{attribute addProperty BoxType "EK1100-0000-0018"}
{attribute addProperty Id "Beckhoff_EM7xxxEK1122Beckhoff_EM7xxxEK1122_7F196951162A_0001_EM7004_0000_9995EM7004_03A980A573692A_0002_EM7004_0000_9996EM7004_78FC6930920115A_0003_EM7004_0000_9997EM7004_78FC6930920115A_0004_EM7004_0000_0016EM7004_A38AEEB0952119A_0005_EM7004_0000_0017EM7004_1DEDE50054468A_0006_EM7004_0000_0018EM7004_1DEDE50054468"}
{attribute addProperty CRC "2403096270"}
{attribute addProperty SizeInBites "4632"}
{attribute addProperty SizeInBytes "579"}
TYPE Beckhoff_EM7xxx_8F3C56CE EXTENDS EK1100_179A0949 :
STRUCT
	{attribute addProperty Name "Beckhoff_EM7xxxEK1122"}
	Beckhoff_EM7xxxEK1122 : Beckhoff_EM7xxxEK1122_7F196951;
	{attribute addProperty Name "A_0001_EM7004_0000_9995"}
	A_0001_EM7004_0000_9995 : EM7004_03A980A5;
	{attribute addProperty Name "A_0002_EM7004_0000_9996"}
	A_0002_EM7004_0000_9996 : EM7004_78FC6930;
	{attribute addProperty Name "A_0003_EM7004_0000_9997"}
	A_0003_EM7004_0000_9997 : EM7004_78FC6930;
	{attribute addProperty Name "A_0004_EM7004_0000_0016"}
	A_0004_EM7004_0000_0016 : EM7004_A38AEEB0;
	{attribute addProperty Name "A_0005_EM7004_0000_0017"}
	A_0005_EM7004_0000_0017 : EM7004_1DEDE500;
	{attribute addProperty Name "A_0006_EM7004_0000_0018"}
	A_0006_EM7004_0000_0018 : EM7004_1DEDE500;
END_STRUCT
END_TYPE

(* stored: Version 1.2.0.0, ProductVersion 3.1.4024.9
   DUT Beckhoff_EM7xxx_8F3C56CE: Id {3f919d0a-3846-4fa9-ab19-786d1223fd08} *)
